{attribute addProperty BoxType "EL2602-0010-0016"}
{attribute addProperty Id "StatusAT %I*BOOL81"}
{attribute addProperty CRC "3186727238"}
{attribute addProperty SizeInBites "8"}
{attribute addProperty SizeInBytes "1"}
TYPE Inputs_BDF19946 :
STRUCT
	{attribute addProperty Name "Status"}
	Status AT %I* : BOOL;
END_STRUCT
END_TYPE

(* stored: Version 1.2.0.0, ProductVersion 3.1.4024.9
   DUT Inputs_BDF19946: Id {fc28522d-4947-4833-9fe0-4f3ccc408d1e} *)
